// TIA Portal project "babu_multipleswitches1" (V15)

(* hardware
DEVICE "S7-1200 station_1"  S7-1200 Station
   slot 0: "Rack_0"  S7-1200 Rack  Rack  V1.0
   slot 1: "PLC_1"  CPU 1212C DC/DC/DC  6ES7 212-1AE40-0XB0  V4.2
*)

// ===== PLC "PLC_1"  CPU 1212C DC/DC/DC =====

VAR_GLOBAL   // PLC tag table "Tag table_1"
   "S1" AT %M0.0 : Bool;
   "S2" AT %M0.1 : Bool;
   "S3" AT %M0.2 : Bool;
   "S4" AT %M0.3 : Bool;
   "S5" AT %M0.4 : Bool;
   "S6" AT %M0.5 : Bool;
   "L1" AT %Q0.6 : Bool;
   "L2" AT %Q0.7 : Bool;
   "L3" AT %Q1.0 : Bool;
   "L4" AT %Q1.1 : Bool;
   "L5" AT %Q1.2 : Bool;
   "L6" AT %Q1.3 : Bool;
   "L7" AT %Q1.4 : Bool;
   "L8" AT %Q1.5 : Bool;
   "L9" AT %Q1.6 : Bool;
END_VAR

ORGANIZATION_BLOCK "Main"   // OB1, LAD, ProgramCycle
TITLE = "Main Program Sweep (Cycle)"
{ S7_Optimized_Access := 'TRUE' }
VERSION : 0.1
   VAR_INPUT
      Initial_Call : Bool;   // Initial call of this OB
      Remanence : Bool;   // =True, if remanent data are available
   END_VAR
BEGIN

REGION Network 1
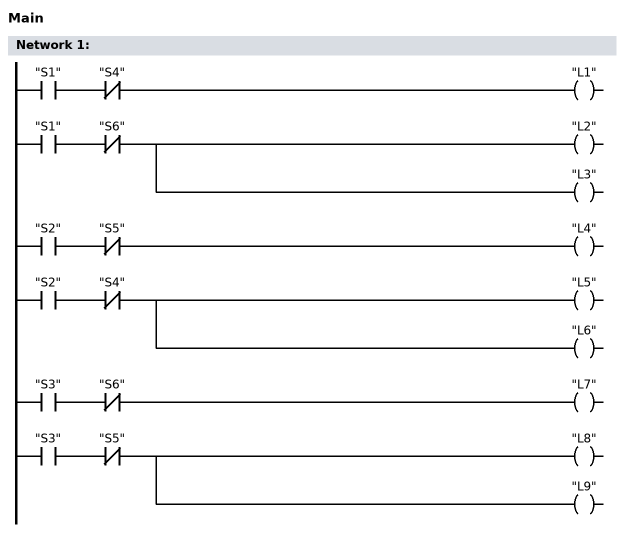
   RUNG wire#powerrail
      Contact( "S1" )
      I_Contact( "S4" )
      Coil( "L1" )
   END_RUNG
   RUNG wire#powerrail
      Contact( "S1" )
      I_Contact( "S6" )
      wire#w1
      Coil( "L2" )
   END_RUNG
   RUNG wire#w1
      Coil( "L3" )
   END_RUNG
   RUNG wire#powerrail
      Contact( "S2" )
      I_Contact( "S5" )
      Coil( "L4" )
   END_RUNG
   RUNG wire#powerrail
      Contact( "S2" )
      I_Contact( "S4" )
      wire#w2
      Coil( "L5" )
   END_RUNG
   RUNG wire#w2
      Coil( "L6" )
   END_RUNG
   RUNG wire#powerrail
      Contact( "S3" )
      I_Contact( "S6" )
      Coil( "L7" )
   END_RUNG
   RUNG wire#powerrail
      Contact( "S3" )
      I_Contact( "S5" )
      wire#w3
      Coil( "L8" )
   END_RUNG
   RUNG wire#w3
      Coil( "L9" )
   END_RUNG
   // the same network as SCL:
   "L1" := "S1" AND NOT "S4";
   "L2" := "S1" AND NOT "S6";
   "L3" := "L2";
   "L4" := "S2" AND NOT "S5";
   "L5" := "S2" AND NOT "S4";
   "L6" := "L5";
   "L7" := "S3" AND NOT "S6";
   "L8" := "S3" AND NOT "S5";
   "L9" := "L8";
END_REGION
END_ORGANIZATION_BLOCK